FUNCTION_BLOCK FB_Input EXTENDS FB_Base
VAR_INPUT
	bAT_bHardwareLink	AT %I*	:	BOOL; // hardware link
END_VAR
VAR_OUTPUT
END_VAR
VAR
	
END_VAR

//FB_Init ist immer implizit verfügbar und wird primär für die Initialisierung verwendet.
//Der Rückgabewert wird nicht ausgewertet. Für gezielte Einflussnahme können Sie
//die Methoden explizit deklarieren und darin mit dem Standard-Initialisierungscode 
//zusätzlichen Code bereitstellen. Sie können den Rückgabewert auswerten.
METHOD FB_Init: BOOL
VAR_INPUT    
	bInitRetains					: BOOL; 					// TRUE: Die Retain-Variablen werden initialisiert (Reset warm / Reset kalt)    
	bInCopyCode						: BOOL;  					// TRUE: Die Instanz wird danach in den Kopiercode kopiert (Online-Change)
	
	I_Name                : STRING;         //  Name
	I_ID                  : UINT;            // ID
END_VAR
END_METHOD

END_FUNCTION_BLOCK

(* stored: Version 1.1.0.1, ProductVersion 3.1.4026.18
   POU FB_Input: Id {03a6797d-89e6-4bde-a671-dac2f9ab8585}, SpecialFunc None
   Folder 01 Properties: Id {dd12400f-aed7-4dfb-b4cb-d45c40bffe5f}
   Folder 02 Methodes: Id {ddadb740-76eb-481d-b099-2fbd7a9a1f63}
   Method FB_Init: Id {4e017715-16ee-49cc-b11c-5f9f51604256} *)
